VAR_GLOBAL
	(*------ Variable in the database ------*)
	rTemp1 : REAL;
	rTemp2 : REAL;
	rTemp3 : REAL;
	bToggle : INT;
	sComment: STRING;
	
	tStoreVar : TIME := T#5000MS;
	tRetrieveVar: TIME := T#5000MS;
	stRecord : ST_Record;
	nID: T_ULARGE_INTEGER;
END_VAR

(* stored: Version 1.1.0.1, ProductVersion 3.1.4020.6
   GVL GVL: Id {0de0043b-907d-45a3-a9f1-a04d3d44455f} *)
